// Mitsubishi GX Works2 project: Main (10)   PLC: FX3G

// global labels: Global1
VAR_GLOBAL
  start AT X007 : BOOL;
  During_day AT Y000 : BOOL;
  Emergency_b AT X005 : BOOL;
  Not_day_finish AT M30 : BOOL;
  Day_finish_protein AT M19 : BOOL;
  Day_finish_Classic AT M18 : BOOL;
  Classic_check AT M4 : BOOL;
  Protein_check AT M5 : BOOL;
  Inv_good AT M3 : BOOL;
  Is_Classic AT M2 : BOOL;
  X_0 AT X000 : BOOL;
  x0_isOn AT M25 : BOOL;
  move_to_bake AT X002 : BOOL;
  Not_finish_Pack_1 AT M40 : BOOL;
  finished_mixing_classic AT M6 : BOOL;
  finished_mixing_protein AT M7 : BOOL;
  start_baking_classic AT M8 : BOOL;
  start_baking_protein AT M9 : BOOL;
  Is_Protein AT M21 : BOOL;
  analog_input1 AT D8280 : INT;
  NumOfPacks AT D1111 : REAL;
  analog_output AT D8282 : INT;
  Job_3 AT X003 : BOOL;
  y_3 AT Y003 : BOOL;
  timer_when_mixing AT TS1 : BOOL;
  finish_bake_protein AT TS14 : BOOL;
  finish_bake_classic AT TS13 : BOOL;
  Y_2 AT Y002 : BOOL;
  M_100 AT M100 : BOOL;
  blink_Y2 AT TS30 : BOOL;
  blink_Y1 AT TS31 : BOOL;
  Y_1 AT Y001 : BOOL;
  X_6 AT X006 : BOOL;
  CS_1 AT CS1 : BOOL;
  Y_4 AT Y004 : BOOL;
  normalization AT E400 : REAL;
  const_1 AT E5.0 : REAL;
  const_2 AT E10.0 : REAL;
  Oat_inv AT D4444 : REAL;
  Classic_Oat_need AT E400.0 : REAL;
  Protein_Powder_inv AT D5555 : REAL;
  Classic_Protein_need AT E160.0 : REAL;
  Honey_inv AT D6666 : REAL;
  Classic_Honey_need AT E120.0 : REAL;
  Protein_Oat_need AT E240.0 : REAL;
  Protein_ProteinPowder_need AT E340.0 : REAL;
  Protein_Honey_need AT E160.0 : REAL;
  TC AT TC1 : BOOL;
END_VAR
VAR_GLOBAL CONSTANT
  TIMER_MIXING : INT := 50;
END_VAR
VAR_GLOBAL
  BakingClassic AT TC13 : BOOL;
END_VAR
VAR_GLOBAL CONSTANT
  bakingClassic_40 : INT := 40;
END_VAR
VAR_GLOBAL
  BakingProtein AT TC14 : BOOL;
END_VAR
VAR_GLOBAL CONSTANT
  bakingProtein_50 : INT := 50;
END_VAR
VAR_GLOBAL
  Start_blink2 AT TC30 : BOOL;
END_VAR
VAR_GLOBAL CONSTANT
  blink : INT := 5;
END_VAR
VAR_GLOBAL
  Start_blink1 AT TC31 : BOOL;
END_VAR
VAR_GLOBAL CONSTANT
  blink2 : INT := 5;
END_VAR
VAR_GLOBAL
  cc_1 AT CC1 : BOOL;
END_VAR
VAR_GLOBAL CONSTANT
  counter8 : INT := 8;
END_VAR
VAR_GLOBAL
  addingPack AT E0.1 : REAL;
  mulFourty AT E400.0 : REAL;
  const_0 AT E0.0 : REAL;
  const_3 AT E6.0 : REAL;
END_VAR

// task Task_01 (event TRUE, interval 0, priority 31): POU_01

PROGRAM POU_01
(* structured ladder/FBD written out as ST: instructions are called as NAME(EN, inputs, outputs); _pN, _eN, _tN stand for wires *)
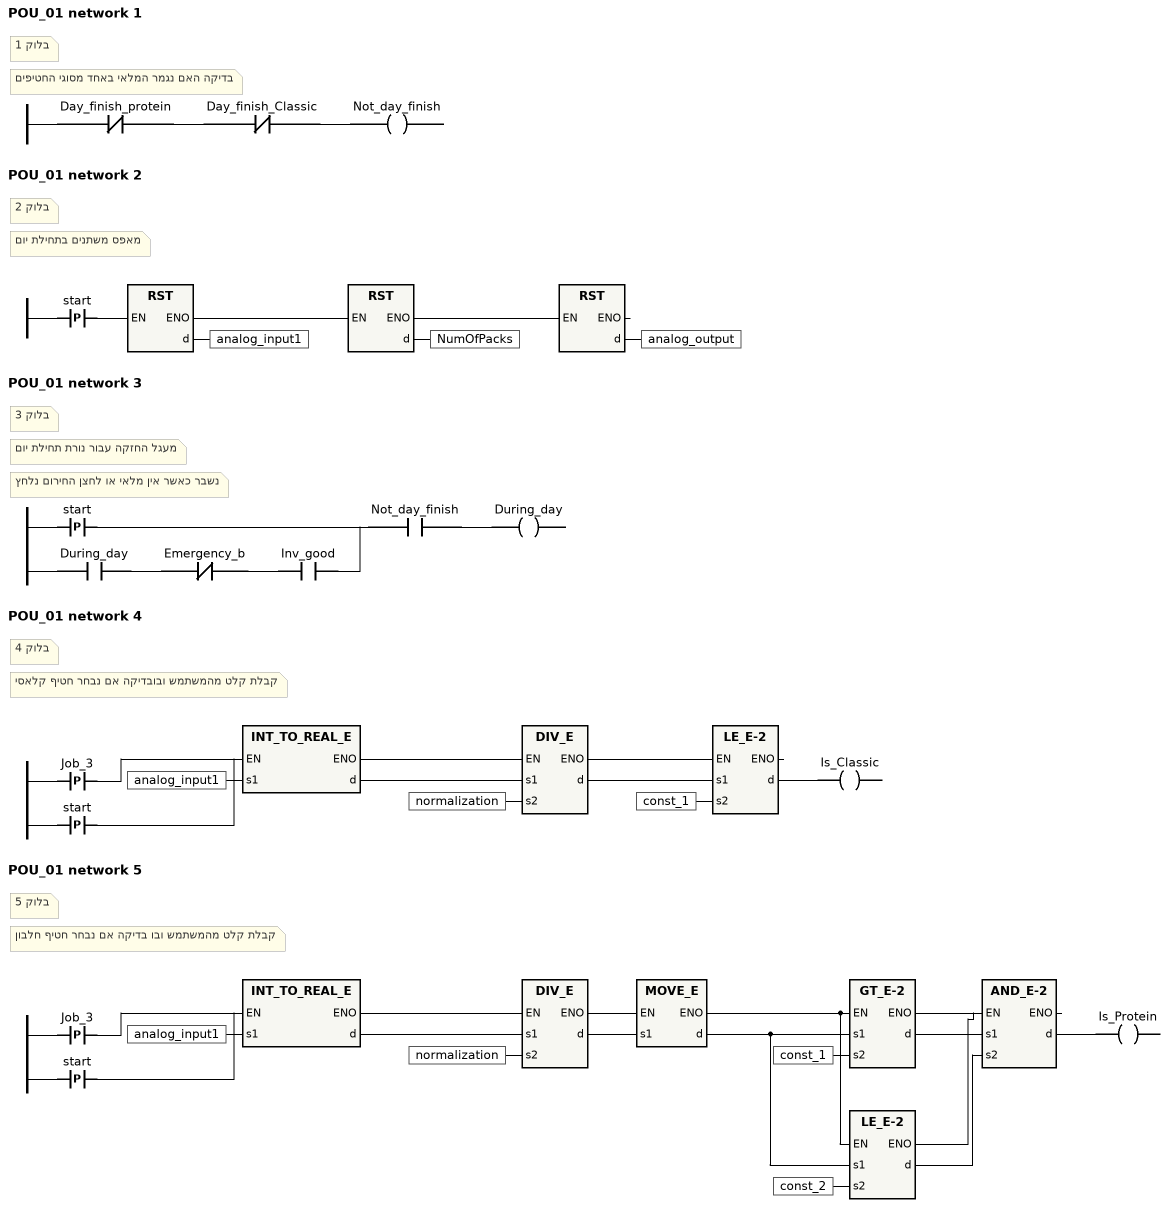
(* network 1 *)
(* בלוק 1 *)
(* בדיקה האם נגמר המלאי באחד מסוגי החטיפים *)
Not_day_finish := NOT Day_finish_protein AND NOT Day_finish_Classic;
(* network 2 *)
(* בלוק 2 *)
(* מאפס משתנים בתחילת יום *)
_e1 := RST(LDP(TRUE, start), analog_input1);
_e2 := RST(_e1, NumOfPacks);
RST(_e2, analog_output);
(* network 3 *)
(* בלוק 3 *)
(* מעגל החזקה עבור נורת תחילת יום *)
(* נשבר כאשר אין מלאי או לחצן החירום נלחץ *)
During_day := (LDP(TRUE, start) OR (During_day AND NOT Emergency_b AND Inv_good)) AND Not_day_finish;
(* network 4 *)
(* בלוק 4 *)
(* קבלת קלט מהמשתמש ובובדיקה אם נבחר חטיף קלאסי *)
_e2 := INT_TO_REAL_E(LDP(TRUE, Job_3) OR LDP(TRUE, start), analog_input1, _t1);
_e4 := DIV_E(_e2, _t1, normalization, _t3);
LE_E(_e4, _t3, const_1, _t5);
Is_Classic := _t5;
(* network 5 *)
(* בלוק 5 *)
(* קבלת קלט מהמשתמש ובו בדיקה אם נבחר חטיף חלבון *)
_e2 := INT_TO_REAL_E(LDP(TRUE, Job_3) OR LDP(TRUE, start), analog_input1, _t1);
_e4 := DIV_E(_e2, _t1, normalization, _t3);
_e6 := MOVE_E(_e4, _t3, _t5);
_e8 := GT_E(_e6, _t5, const_1, _t7);
_e10 := LE_E(_e6, _t5, const_2, _t9);
AND_E(_e8 OR _e10, _t7, _t9, _t11);
Is_Protein := _t11;
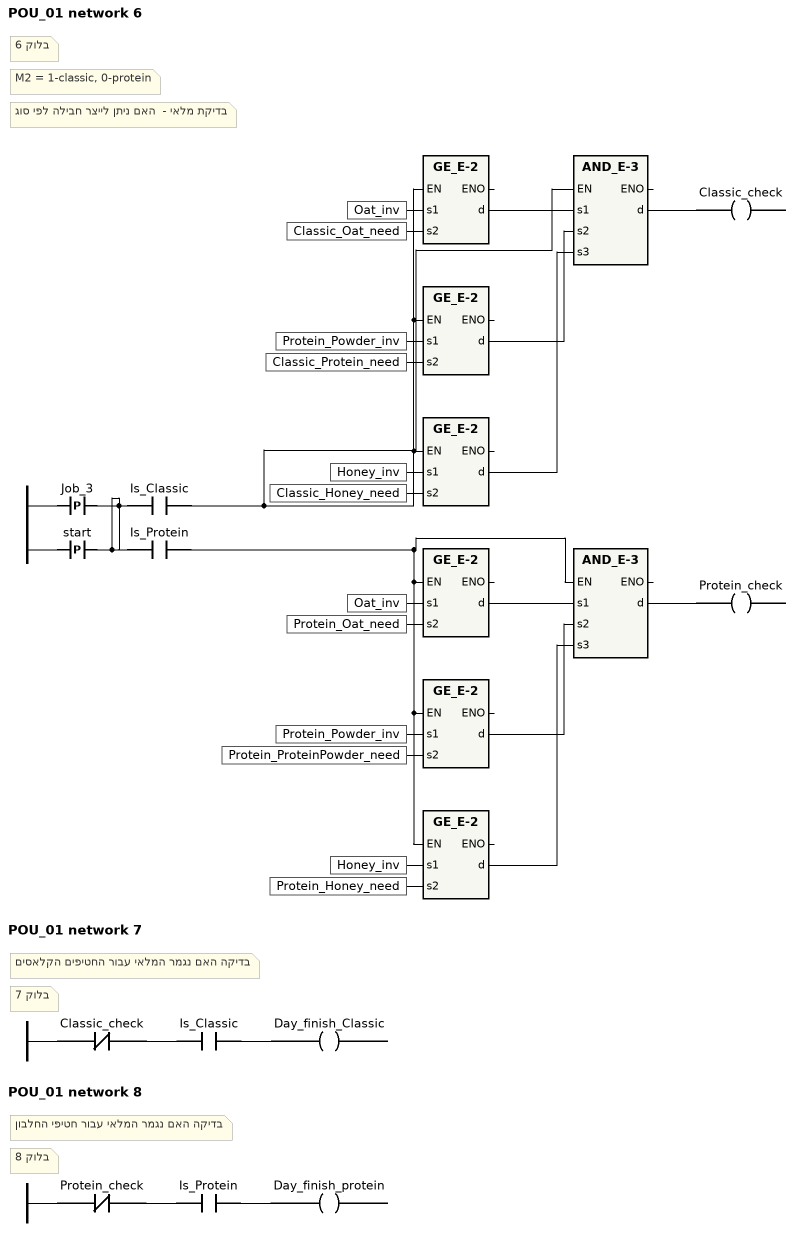
(* network 6 *)
(* בלוק 6 *)
(* M2 = 1-classic, 0-protein *)
(* בדיקת מלאי -  האם ניתן לייצר חבילה לפי סוג *)
_p1 := LDP(TRUE, Job_3) OR LDP(TRUE, start);
_p2 := _p1 AND Is_Classic;
GE_E(_p2, Oat_inv, Classic_Oat_need, _t3);
GE_E(_p2, Protein_Powder_inv, Classic_Protein_need, _t4);
GE_E(_p2, Honey_inv, Classic_Honey_need, _t5);
AND_E(_p2, _t3, _t4, _t5, _t6);
Classic_check := _t6;
_p7 := _p1 AND Is_Protein;
GE_E(_p7, Oat_inv, Protein_Oat_need, _t8);
GE_E(_p7, Protein_Powder_inv, Protein_ProteinPowder_need, _t9);
GE_E(_p7, Honey_inv, Protein_Honey_need, _t10);
AND_E(_p7, _t8, _t9, _t10, _t11);
Protein_check := _t11;
(* network 7 *)
(* בדיקה האם נגמר המלאי עבור החטיפים הקלאסים *)
(* בלוק 7 *)
Day_finish_Classic := NOT Classic_check AND Is_Classic;
(* network 8 *)
(* בדיקה האם נגמר המלאי עבור חטיפי החלבון *)
(* בלוק 8 *)
Day_finish_protein := NOT Protein_check AND Is_Protein;
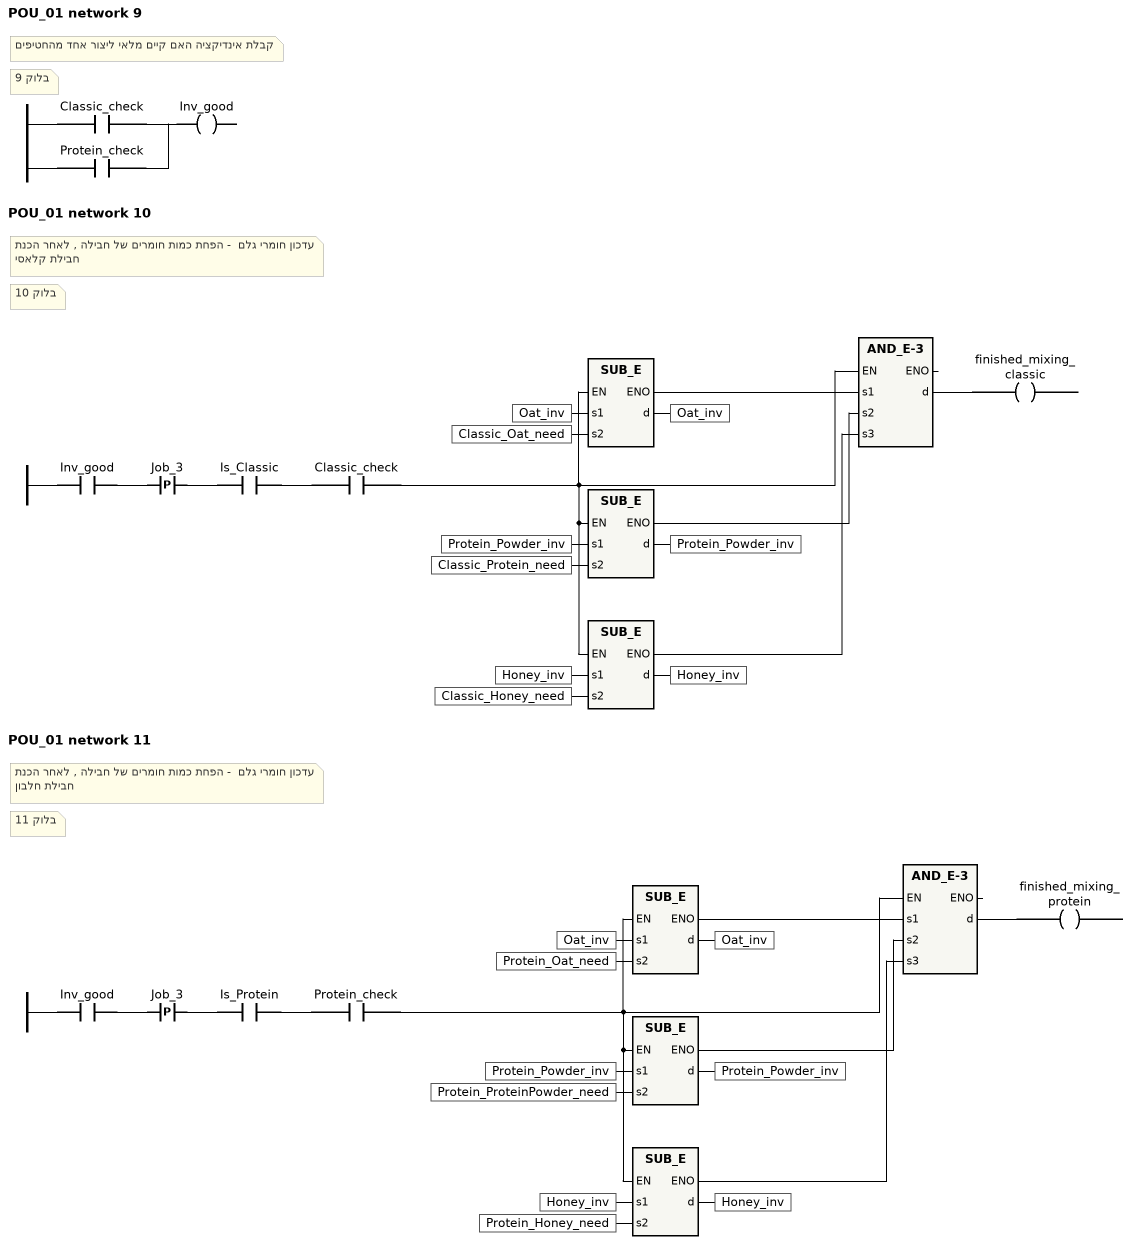
(* network 9 *)
(* קבלת אינדיקציה האם קיים מלאי ליצור אחד מהחטיפים *)
(* בלוק 9 *)
Inv_good := Classic_check OR Protein_check;
(* network 10 *)
(* עדכון חומרי גלם  - הפחת כמות חומרים של חבילה , לאחר הכנת חבילת קלאסי *)
(* בלוק 10 *)
_p1 := Inv_good AND LDP(TRUE, Job_3) AND Is_Classic AND Classic_check;
_e2 := SUB_E(_p1, Oat_inv, Classic_Oat_need, Oat_inv);
_e3 := SUB_E(_p1, Protein_Powder_inv, Classic_Protein_need, Protein_Powder_inv);
_e4 := SUB_E(_p1, Honey_inv, Classic_Honey_need, Honey_inv);
AND_E(_p1, _e2, _e3, _e4, _t5);
finished_mixing_classic := _t5;
(* network 11 *)
(* עדכון חומרי גלם  - הפחת כמות חומרים של חבילה , לאחר הכנת חבילת חלבון *)
(* בלוק 11 *)
_p1 := Inv_good AND LDP(TRUE, Job_3) AND Is_Protein AND Protein_check;
_e2 := SUB_E(_p1, Oat_inv, Protein_Oat_need, Oat_inv);
_e3 := SUB_E(_p1, Protein_Powder_inv, Protein_ProteinPowder_need, Protein_Powder_inv);
_e4 := SUB_E(_p1, Honey_inv, Protein_Honey_need, Honey_inv);
AND_E(_p1, _e2, _e3, _e4, _t5);
finished_mixing_protein := _t5;
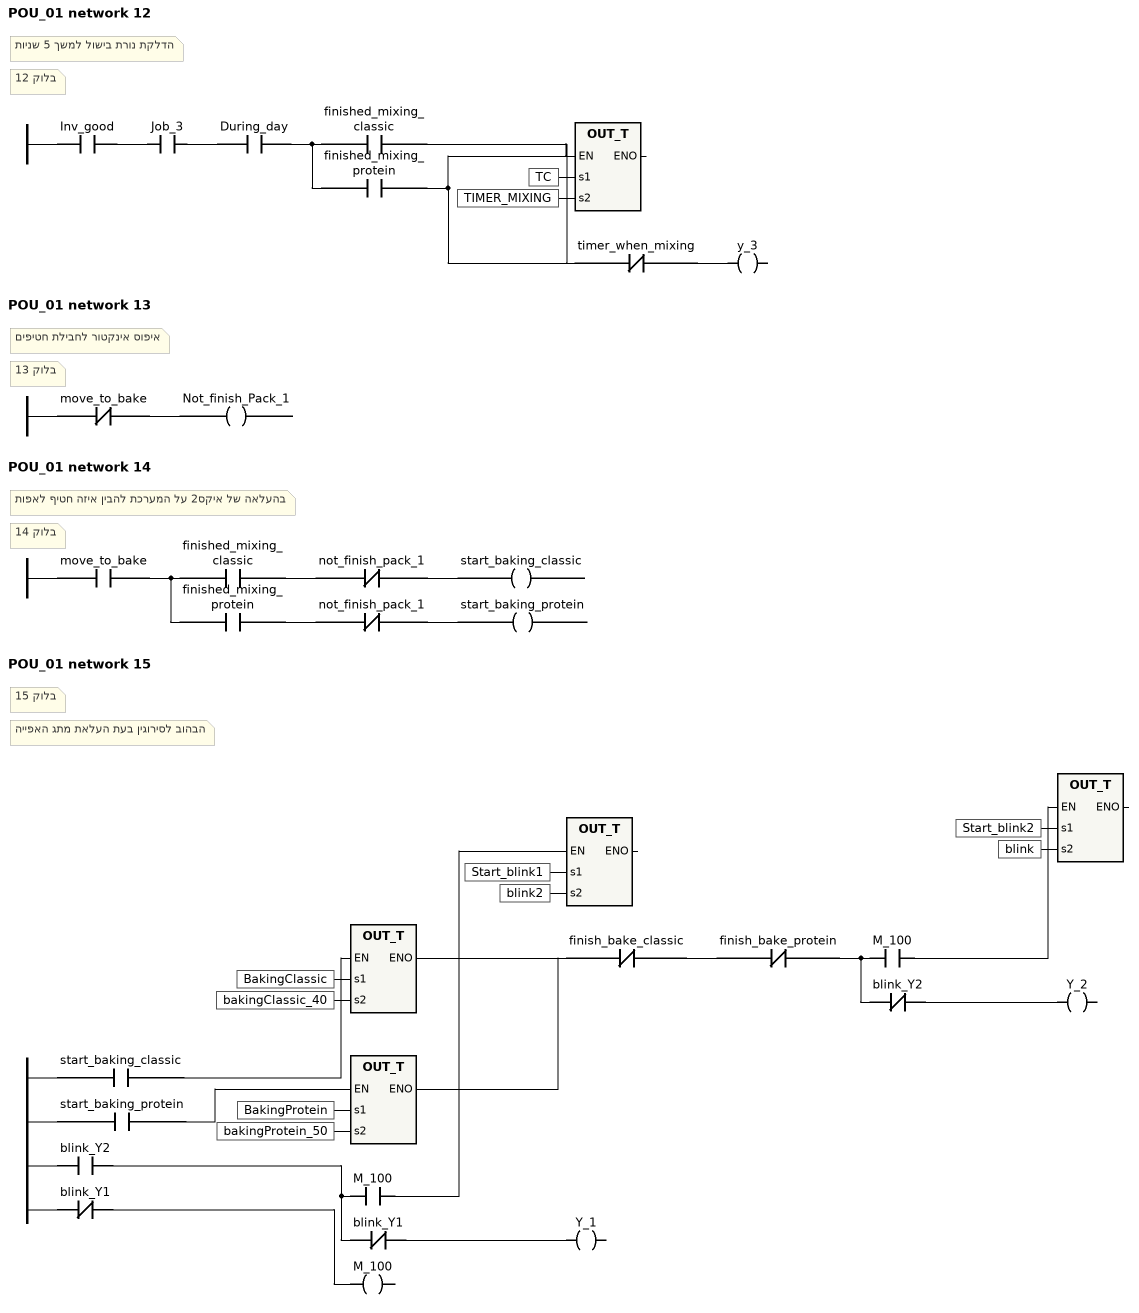
(* network 12 *)
(* הדלקת נורת בישול למשך 5 שניות *)
(* בלוק 12 *)
_p1 := Inv_good AND Job_3 AND During_day;
_p2 := (_p1 AND finished_mixing_classic) OR (_p1 AND finished_mixing_protein);
y_3 := _p2 AND NOT timer_when_mixing;
OUT_T(_p2, TC, TIMER_MIXING);
(* network 13 *)
(* איפוס אינקטור לחבילת חטיפים *)
(* בלוק 13 *)
Not_finish_Pack_1 := NOT move_to_bake;
(* network 14 *)
(* בהעלאה של איקס2 על המערכת להבין איזה חטיף לאפות *)
(* בלוק 14 *)
start_baking_classic := move_to_bake AND finished_mixing_classic AND NOT not_finish_pack_1;
start_baking_protein := move_to_bake AND finished_mixing_protein AND NOT not_finish_pack_1;
(* network 15 *)
(* בלוק 15 *)
(* הבהוב לסירוגין בעת העלאת מתג האפייה *)
_e1 := OUT_T(start_baking_classic, BakingClassic, bakingClassic_40);
_e2 := OUT_T(start_baking_protein, BakingProtein, bakingProtein_50);
_p3 := ((_e1 OR _e2) AND NOT finish_bake_classic) AND NOT finish_bake_protein;
OUT_T(_p3 AND M_100, Start_blink2, blink);
Y_2 := _p3 AND NOT blink_Y2;
OUT_T(blink_Y2 AND M_100, Start_blink1, blink2);
Y_1 := blink_Y2 AND NOT blink_Y1;
M_100 := NOT blink_Y1;
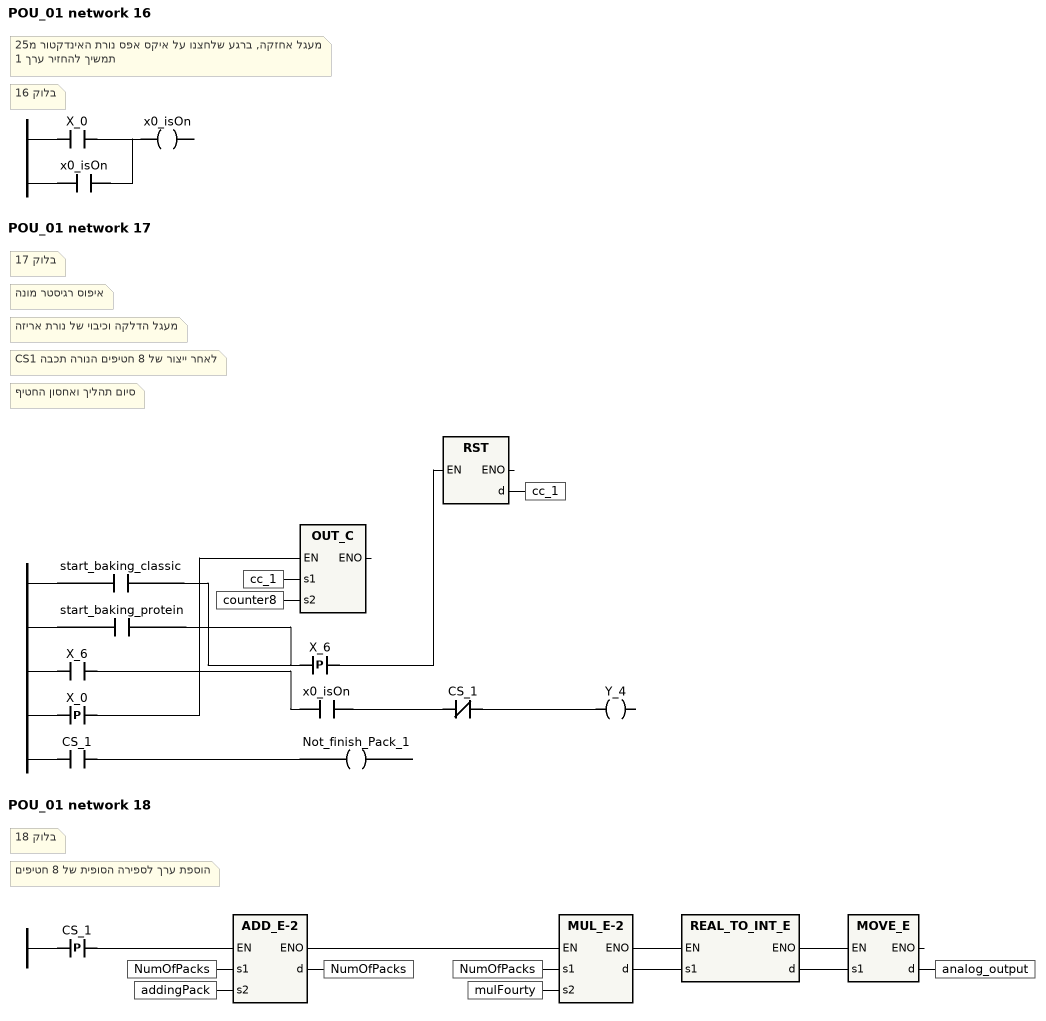
(* network 16 *)
(* מעגל אחזקה, ברגע שלחצנו על איקס אפס נורת האינדקטור מ25 תמשיך להחזיר ערך 1 *)
(* בלוק 16 *)
x0_isOn := X_0 OR x0_isOn;
(* network 17 *)
(* בלוק 17 *)
(* איפוס רגיסטר מונה *)
(* מעגל הדלקה וכיבוי של נורת אריזה *)
(* לאחר ייצור של 8 חטיפים הנורה תכבה CS1 *)
(* סיום תהליך ואחסון החטיף *)
RST((start_baking_classic OR start_baking_protein) AND LDP(TRUE, X_6), cc_1);
Y_4 := X_6 AND x0_isOn AND NOT CS_1;
OUT_C(LDP(TRUE, X_0), cc_1, counter8);
Not_finish_Pack_1 := CS_1;
(* network 18 *)
(* בלוק 18 *)
(* הוספת ערך לספירה הסופית של 8 חטיפים *)
_e1 := ADD_E(LDP(TRUE, CS_1), NumOfPacks, addingPack, NumOfPacks);
_e3 := MUL_E(_e1, NumOfPacks, mulFourty, _t2);
_e5 := REAL_TO_INT_E(_e3, _t2, _t4);
MOVE_E(_e5, _t4, analog_output);
END_PROGRAM
